FUNCTION_BLOCK FB_FT_TN8 (* Basic Function Block Type *)
  (* Standard: 61499-2 *)
  (* Version 0.0, 2011-08-30, 4DIAC-IDE, 4DIAC-Consortium *)
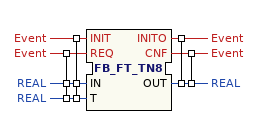
  EVENT_INPUT
    INIT WITH IN, T; (* Initialization Request *)
    REQ WITH IN, T; (* Normal Execution Request *)
  END_EVENT
  EVENT_OUTPUT
    INITO WITH OUT; (* Initialization Confirm *)
    CNF WITH OUT; (* Execution Confirmation *)
  END_EVENT
  VAR_INPUT
    IN : REAL; (* Input event qualifier *)
    T : REAL;
  END_VAR
  VAR_OUTPUT
    OUT : REAL; (* Output event qualifier *)
  END_VAR
  VAR
    length : INT := 8; (* Internal Variable *)
    X : ARRAY [0..7] OF REAL; (* Internal Variable *)
    cnt : INT; (* Internal Variable *)
    last : TIME; (* Internal Variable *)
    tx : TIME; (* Internal Variable *)
  END_VAR
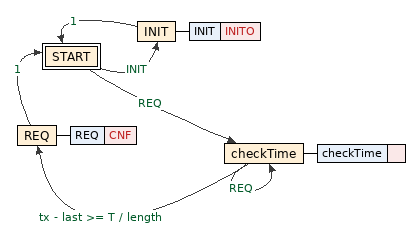
  EC_STATES
    START; (* Initial State *)
    INIT : INIT -> INITO; (* Initialization *)
    REQ : REQ -> CNF; (* Normal execution *)
    checkTime : checkTime;
  END_STATES
  EC_TRANSITIONS
    START TO INIT := INIT;
    INIT TO START := 1;
    REQ TO START := 1;
    START TO checkTime := REQ;
    checkTime TO checkTime := REQ;
    checkTime TO REQ := tx - last >= T / length;
  END_TRANSITIONS
  ALGORITHM INIT IN ST: (* Initialization algorithm *)
X[cnt] := IN;
last := TIME();
  END_ALGORITHM
  ALGORITHM REQ IN ST: (* Normally executed algorithm *)
IF cnt = length - 1 THEN
  cnt := 0;
ELSE
  cnt := cnt + 1;
END_IF;

OUT := X[cnt];
X[cnt] := IN;
last := tx;
  END_ALGORITHM
  ALGORITHM checkTime IN ST: (* ALG *)
tx :=TIME();
  END_ALGORITHM
END_FUNCTION_BLOCK
